{attribute 'qualified_only'}
VAR_GLOBAL
	xCorrectHeight : BOOL;
	rZeroOffset : REAL;
	rActual: REAL;
	rDesiredHeight: REAL;
END_VAR

(* stored: Version 1.1.0.1, ProductVersion 3.1.4024.11
   GVL G_HeightCorrection: Id {570bc1fa-d823-42f1-b5de-c19e1ec1e040} *)
